INTERFACE ITF_AutoStructCommand

PROPERTY Connect : String(50)
GET
END_GET
SET
END_SET
END_PROPERTY

PROPERTY Error : BOOL
GET
END_GET
END_PROPERTY

METHOD ErrorClear : BOOL
VAR_INPUT
END_VAR
END_METHOD

METHOD FB_init : BOOL
VAR_INPUT
	bInitRetains : BOOL; // if TRUE, the retain variables are initialized (warm start / cold start)
	bInCopyCode : BOOL;  // if TRUE, the instance afterwards gets moved into the copy code (online change)
END_VAR
END_METHOD

METHOD HaltStepContiune : BOOL
VAR_INPUT
END_VAR
END_METHOD

METHOD Initialization : BOOL
VAR_INPUT
	_Testmode	:BOOL;
END_VAR
END_METHOD

PROPERTY NoEntry : BOOL	//不允許進入
GET
END_GET
END_PROPERTY

METHOD Pause : BOOL
VAR_INPUT
END_VAR
END_METHOD

METHOD Process : BOOL
VAR_INPUT
	bHlatMode	:BOOL;
END_VAR
END_METHOD

PROPERTY Status : STRING(50)
GET
END_GET
END_PROPERTY

END_INTERFACE

(* stored: Version 1.1.0.1, ProductVersion 3.1.4024.16
   Itf ITF_AutoStructCommand: Id {50094617-8a33-40db-8fe0-6b5f4573bb55}
   Property Connect: Id {96de4d5a-759b-431e-89f8-6aec36ea2ef7}
   Get Get: Id {37e08c77-94e0-4f9e-8afc-81f872cfbfa2}
   Set Set: Id {22f93a74-3782-46a0-b33d-8d5361f3a555}
   Property Error: Id {33c807c2-98a2-47ab-9d0a-e17d4899fe09}
   Get Get: Id {008099b1-37d5-4cda-819e-3df27be2515d}
   Method ErrorClear: Id {23cbff6e-02ff-425b-a4bf-485ff535cad9}
   Method FB_init: Id {2f417aaf-5c67-46a9-8a73-59b1143c43b4}
   Method HaltStepContiune: Id {694d5575-5e40-46a3-b62d-efb0b44def6b}
   Method Initialization: Id {901fff7e-347a-476f-a2ae-3c276b2a61e3}
   Property NoEntry: Id {4ee6eb86-7e84-44b8-a4ff-cf9f9ec60f29}
   Get Get: Id {2ee615cc-e1f2-45d6-8b66-fc3b444a25ca}
   Method Pause: Id {ab1cf2db-915d-447b-85e6-ce6e7d72cf6d}
   Method Process: Id {97fe5338-3003-4b5d-bcfa-48b4d5d246f6}
   Property Status: Id {42473ac0-2151-4c46-949a-b74ee7f04eb4}
   Get Get: Id {4bd8df53-b551-4441-9b1a-ccaba4465320} *)
